FUNCTION_BLOCK E_INIT_CHK (* Sends INIT event the first time a REQ event arrives and a NOINIT event for every subsequent REQ event. *)
  (* Standard: 61499-2 *)
  (* Version 0.0, 2017-06-17, 4DIAC-IDE, 4DIAC-Consortium *)
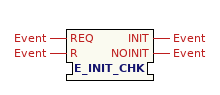
  EVENT_INPUT
    REQ; (* Normal Execution Request *)
    R; (* Reset *)
  END_EVENT
  EVENT_OUTPUT
    INIT; (* Initialization *)
    NOINIT; (* No initialization *)
  END_EVENT
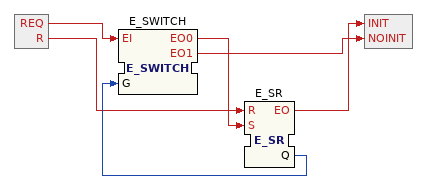
  FBS
    E_SR : E_SR;
    E_SWITCH : E_SWITCH;
  END_FBS
  EVENT_CONNECTIONS
    REQ TO E_SWITCH.EI;
    R TO E_SR.R;
    E_SWITCH.EO0 TO E_SR.S;
    E_SR.EO TO INIT;
    E_SWITCH.EO1 TO NOINIT;
  END_CONNECTIONS
  DATA_CONNECTIONS
    E_SR.Q TO E_SWITCH.G;
  END_CONNECTIONS
END_FUNCTION_BLOCK
